// TIA Portal V15.1 export
// export: Created 2020-06-12T07:35:49.0849609Z, ExportSetting None, DisplayName Totally Integrated Automation Portal, DisplayVersion V15.1, DisplayName TIA Portal Openness, DisplayVersion V15.1, DisplayName STEP 7 Professional, DisplayVersion V15.1, DisplayName STEP 7 Safety, DisplayVersion V15.1, DisplayName WinCC Advanced, DisplayVersion V15.1
FUNCTION "HOOD_call" : Void   // FC85, FBD
TITLE = Hood carriage call
{ S7_Optimized_Access := 'TRUE' }
// stored: SetENOAutomatically False
BEGIN

REGION Network 1: Hood Movement
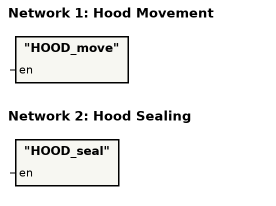
   "HOOD_move"();
END_REGION

REGION Network 2: Hood Sealing
   "HOOD_seal"();
END_REGION
END_FUNCTION
